FUNCTION_BLOCK ConveyorControlUnit
VAR_IN_OUT
	conveyors : ARRAY[*] OF POINTER TO ConveyorSC;
END_VAR
VAR
	firstConveyor : DINT;
	lastConveyor : DINT;
	
	spoolTimer : TON;
	i : DINT := 1;
END_VAR
VAR CONSTANT
	spoolSpacing : TIME := T#100MS;
END_VAR

firstConveyor := LOWER_BOUND(conveyors, 1);
lastConveyor := UPPER_BOUND(conveyors, 1);

//use one or the other, not both
linkCompute();
//cyclicCompute();

spoolTimer(IN:= , PT:= spoolSpacing, Q=> , ET=> );
spoolTimer.IN := TRUE;
IF
	(conveyors[i]^.requestedMode = ConveyorMode.FORWARD OR conveyors[i]^.requestedMode = ConveyorMode.BACKWARD) AND //conveyor requests motion
	conveyors[i]^.requestedMode <> conveyors[i]^.trueMode AND //conveyor request differs from current operation
	spoolTimer.Q //ready to spool
THEN
	//spool up conveyor
	i := (i + 1) MOD (lastConveyor - firstConveyor + 1) + 1;
	spoolTimer.IN := FALSE;
END_IF

METHOD PRIVATE cyclicCompute : BOOL
VAR
	i : INT;
END_VAR
(*
cyclic computation method
if the last conveyor has the highest priority in a long link, it will take several cycles to reach the other end
*)
(*
FOR i:=numConveyors TO 1 BY -1 DO
	IF NOT conveyors[i]^.IsOccupied THEN
		//turn conveyor off, but do not change request mode
		conveyors[i]^.setMode(ConveyorMode.IDLE);
		CONTINUE;
	END_IF
	
	//conveyor is occupied:
	IF i = numConveyors THEN //no next conveyor
		conveyors[i]^.setMode( MAX(conveyors[i]^.requestedMode, conveyors[i-1]^.trueMode) );
	
	ELSIF i < numConveyors AND i > 1 THEN
		
		IF conveyors[i+1]^.IsOccupied THEN //next conveyor is occupied
			conveyors[i]^.setMode( MAX(conveyors[i+1]^.trueMode, conveyors[i]^.requestedMode) );
		END_IF
		
	END_IF
	
END_FOR
*)
END_METHOD

METHOD PRIVATE linkCompute : BOOL
VAR
	i : DINT;
	j : DINT;
	
	linkStart : DINT := -1;
	linkEnd : DINT := -1;
	
	priorityInLink : ConveyorMode;
END_VAR
(*
link interation method 
slower, but will correctly set all operations every cycle
*)
FOR i:=LOWER_BOUND(conveyors, 1) TO UPPER_BOUND(conveyors, 1) BY 1 DO
	IF conveyors[i]^.IsOccupied THEN
		
		IF linkStart = -1 THEN
			linkStart := i;
		END_IF
		
		priorityInLink := MAX(priorityInLink, conveyors[i]^.requestedMode);
		linkEnd := i;
		
	ELSIF linkStart <> -1 AND linkEnd <> -1 THEN //set all conveyor operations to priorityInLink
		linkEnd := i-1;
		
		FOR j:=linkStart TO linkEnd BY 1 DO
			conveyors[j]^.setMode(priorityInLink);
		END_FOR
		
		linkStart := -1;
		linkEnd := -1;
		priorityInLink := ConveyorMode.IDLE;
		
		CONTINUE;
	END_IF
	
END_FOR

linkEnd := linkEnd - 1; //remove residual increment from for loop's failed iteration
IF linkStart > -1 AND linkEnd > -1 THEN
	FOR j:=linkStart TO linkEnd BY 1 DO
		conveyors[j]^.setMode(priorityInLink);
	END_FOR
END_IF
END_METHOD

END_FUNCTION_BLOCK

(* stored: Version 1.1.0.1, ProductVersion 3.1.4024.11
   POU ConveyorControlUnit: Id {318a19f0-e7ed-42e5-b785-80a2c36ff413}, SpecialFunc None
   Method cyclicCompute: Id {6b6d1f6e-1b21-4dcf-bff4-57c0dd1d2422}
   Method linkCompute: Id {4b47d7ec-4657-4dc5-8694-93a08a021dcf} *)
